(* CoDeSys 2.3 export: MUL_ARM_BASKET_MEMORY.EXP *)

(* POU MUL_ARM_BASKET_MEMORY, LD *)
FUNCTION_BLOCK MUL_ARM_BASKET_MEMORY
VAR_INPUT
	bLoadUnhook:BOOL;
	bLoadHook:BOOL;
	bUnloadUnhook: BOOL;
	bUnloadHook:BOOL;
	bArmDown: BOOL;
	tSignalFilter : TIME;

END_VAR

VAR_OUTPUT
(*	bPreviousZoneSensor2On: BOOL;
	bPreviousZoneSensor1On: BOOL;
	Inhibit: BOOL;*)


	bNoCurrentStationConfirmBasketFlag: BOOL;
	bNoCurrentStationTransferBasketFlag: BOOL;
	bNoNextStationConfirmBasketFlag: BOOL;
END_VAR
VAR

	LoadUnhookConfirmTimer: TON;
	LoadHookConfirmTimer: TON;
	UnloadUnhookConfirmTimer: TON;
	UnloadHookConfirmTimer: TON;
	PowerUpDelayTimer: TON;
	PUDT_Out: BOOL;


	LoadUnhookDIFU: R_TRIG;
	LoadHookDIFU: R_TRIG;
	UnloadUnhookDIFU: R_TRIG;
	UnloadHookDIFU: R_TRIG;
END_VAR
VAR_IN_OUT


	CurrentStationConfirmBasketName:STRING;
	CurrentStationTransferBasketName:STRING;
	NextStationConfirmBasketName:STRING;

END_VAR
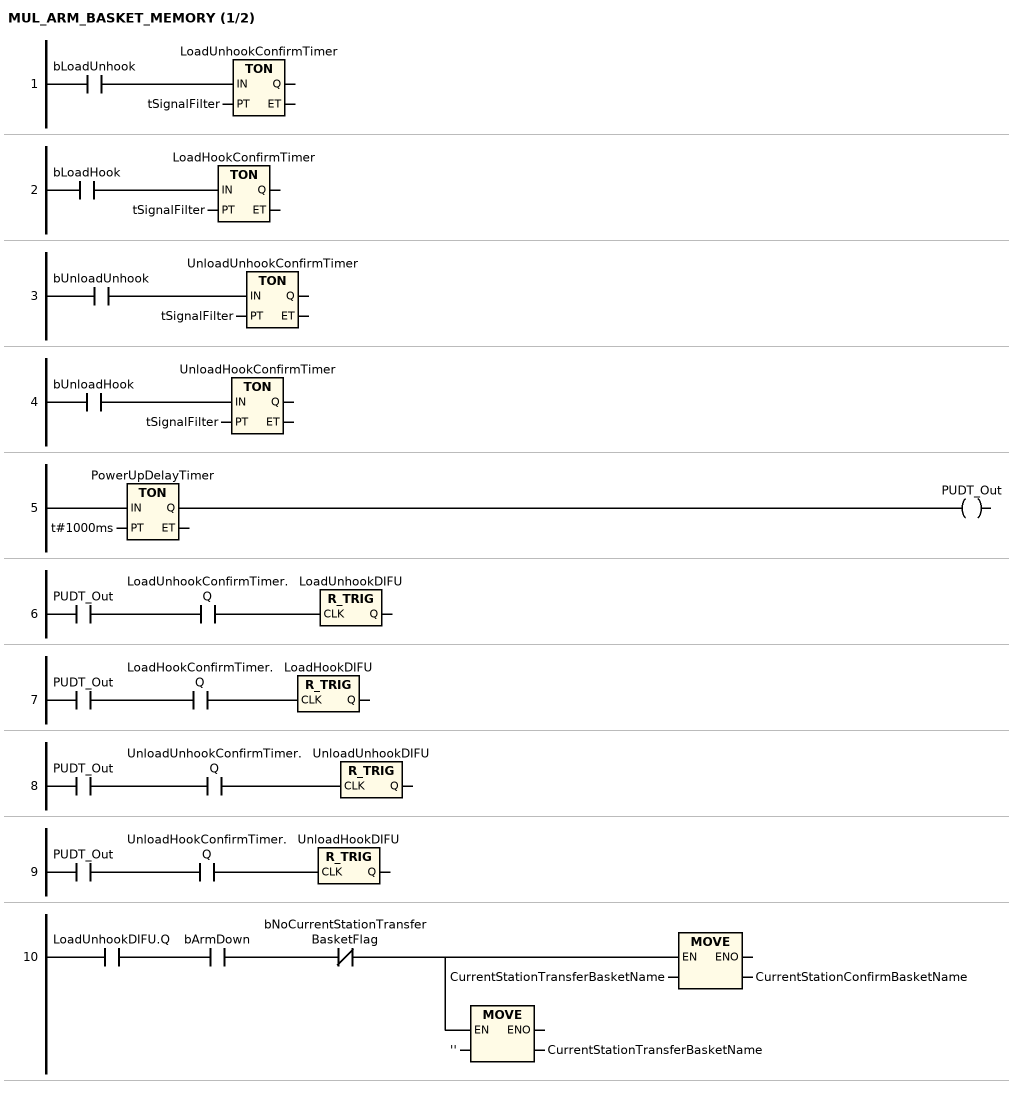
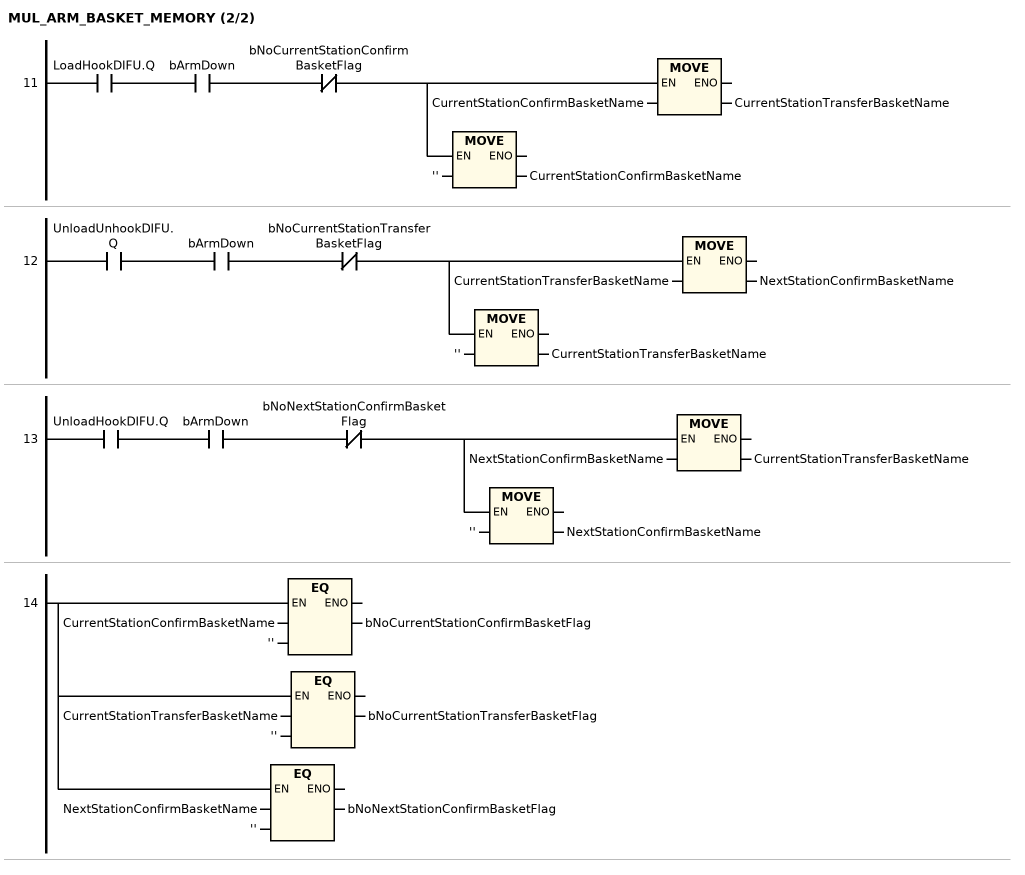
_LD_ (* Ladder Diagram *)
NETWORK 1
	[bLoadUnhook] - LoadUnhookConfirmTimer:TON(IN: *, PT: tSignalFilter)
NETWORK 2
	[bLoadHook] - LoadHookConfirmTimer:TON(IN: *, PT: tSignalFilter)
NETWORK 3
	[bUnloadUnhook] - UnloadUnhookConfirmTimer:TON(IN: *, PT: tSignalFilter)
NETWORK 4
	[bUnloadHook] - UnloadHookConfirmTimer:TON(IN: *, PT: tSignalFilter)
NETWORK 5
	PowerUpDelayTimer:TON(IN: *, PT: t#1000ms) --- (PUDT_Out)
NETWORK 6
	[PUDT_Out] - [LoadUnhookConfirmTimer.Q] - LoadUnhookDIFU:R_TRIG(CLK: *)
NETWORK 7
	[PUDT_Out] - [LoadHookConfirmTimer.Q] - LoadHookDIFU:R_TRIG(CLK: *)
NETWORK 8
	[PUDT_Out] - [UnloadUnhookConfirmTimer.Q] - UnloadUnhookDIFU:R_TRIG(CLK: *)
NETWORK 9
	[PUDT_Out] - [UnloadHookConfirmTimer.Q] - UnloadHookDIFU:R_TRIG(CLK: *)
NETWORK 10
	[LoadUnhookDIFU.Q] - [bArmDown] - [/bNoCurrentStationTransferBasketFlag]
		EN --- MOVE(CurrentStationTransferBasketName) => CurrentStationConfirmBasketName
		EN --- MOVE('') => CurrentStationTransferBasketName
NETWORK 11
	[LoadHookDIFU.Q] - [bArmDown] - [/bNoCurrentStationConfirmBasketFlag]
		EN --- MOVE(CurrentStationConfirmBasketName) => CurrentStationTransferBasketName
		EN --- MOVE('') => CurrentStationConfirmBasketName
NETWORK 12
	[UnloadUnhookDIFU.Q] - [bArmDown] - [/bNoCurrentStationTransferBasketFlag]
		EN --- MOVE(CurrentStationTransferBasketName) => NextStationConfirmBasketName
		EN --- MOVE('') => CurrentStationTransferBasketName
NETWORK 13
	[UnloadHookDIFU.Q] - [bArmDown] - [/bNoNextStationConfirmBasketFlag]
		EN --- MOVE(NextStationConfirmBasketName) => CurrentStationTransferBasketName
		EN --- MOVE('') => NextStationConfirmBasketName
NETWORK 14
	*
		EN --- EQ(CurrentStationConfirmBasketName, '') => bNoCurrentStationConfirmBasketFlag
		EN --- EQ(CurrentStationTransferBasketName, '') => bNoCurrentStationTransferBasketFlag
		EN --- EQ(NextStationConfirmBasketName, '') => bNoNextStationConfirmBasketFlag
_END_LD_
(* the same logic as Structured Text *)
(* Network 1 *)
LoadUnhookConfirmTimer(IN := bLoadUnhook, PT := tSignalFilter);
(* Network 2 *)
LoadHookConfirmTimer(IN := bLoadHook, PT := tSignalFilter);
(* Network 3 *)
UnloadUnhookConfirmTimer(IN := bUnloadUnhook, PT := tSignalFilter);
(* Network 4 *)
UnloadHookConfirmTimer(IN := bUnloadHook, PT := tSignalFilter);
(* Network 5 *)
PowerUpDelayTimer(IN := TRUE, PT := t#1000ms);
PUDT_Out := PowerUpDelayTimer.Q;
(* Network 6 *)
LoadUnhookDIFU(CLK := PUDT_Out AND LoadUnhookConfirmTimer.Q);
(* Network 7 *)
LoadHookDIFU(CLK := PUDT_Out AND LoadHookConfirmTimer.Q);
(* Network 8 *)
UnloadUnhookDIFU(CLK := PUDT_Out AND UnloadUnhookConfirmTimer.Q);
(* Network 9 *)
UnloadHookDIFU(CLK := PUDT_Out AND UnloadHookConfirmTimer.Q);
(* Network 10 *)
IF LoadUnhookDIFU.Q AND bArmDown AND NOT bNoCurrentStationTransferBasketFlag THEN
	CurrentStationConfirmBasketName := CurrentStationTransferBasketName;
	CurrentStationTransferBasketName := '';
END_IF;
(* Network 11 *)
IF LoadHookDIFU.Q AND bArmDown AND NOT bNoCurrentStationConfirmBasketFlag THEN
	CurrentStationTransferBasketName := CurrentStationConfirmBasketName;
	CurrentStationConfirmBasketName := '';
END_IF;
(* Network 12 *)
IF UnloadUnhookDIFU.Q AND bArmDown AND NOT bNoCurrentStationTransferBasketFlag THEN
	NextStationConfirmBasketName := CurrentStationTransferBasketName;
	CurrentStationTransferBasketName := '';
END_IF;
(* Network 13 *)
IF UnloadHookDIFU.Q AND bArmDown AND NOT bNoNextStationConfirmBasketFlag THEN
	CurrentStationTransferBasketName := NextStationConfirmBasketName;
	NextStationConfirmBasketName := '';
END_IF;
(* Network 14 *)
bNoCurrentStationConfirmBasketFlag := CurrentStationConfirmBasketName = '';
bNoCurrentStationTransferBasketFlag := CurrentStationTransferBasketName = '';
bNoNextStationConfirmBasketFlag := NextStationConfirmBasketName = '';
END_FUNCTION_BLOCK
